(* LS Electric XG5000 project: PLC_Playground *)
(* PLC PlaygroundPLC *)

PROGRAM Main (* task: Scan Program *)
VAR
    I_Start AT %IX0.0.0 : BOOL;
    I_Stop AT %IX0.0.1 : BOOL;
    O_Run AT %QX0.0.0 : BOOL;
END_VAR
VAR
    _e1 : R_TRIG;
    _e2 : R_TRIG;
END_VAR

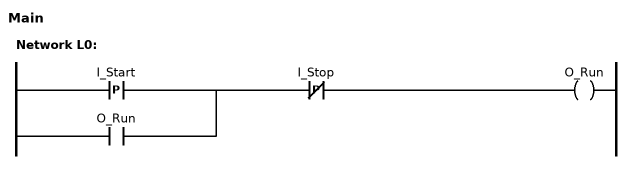
(* Rung L0 *)
_e1(CLK := I_Start);
_e2(CLK := I_Stop);
O_Run := (_e1.Q OR O_Run) AND NOT _e2.Q;
END_PROGRAM

PROGRAM FwdBwdMotor (* task: Scan Program *)
VAR
    I_Btn_Start AT %IX0.0.0 : BOOL;
    I_Btn_Stop AT %IX0.0.1 : BOOL;
    I_Sel_Direction AT %IX0.0.2 : BOOL;
    M_Is_Fwd AT %MX1 : BOOL := 1;
    M_Is_Moving AT %MX0 : BOOL := 0;
    O_Move_Bwd AT %QX0.0.1 : BOOL;
    O_Move_Fwd AT %QX0.0.0 : BOOL;
END_VAR
VAR
    _e1 : R_TRIG;
    _e2 : R_TRIG;
END_VAR

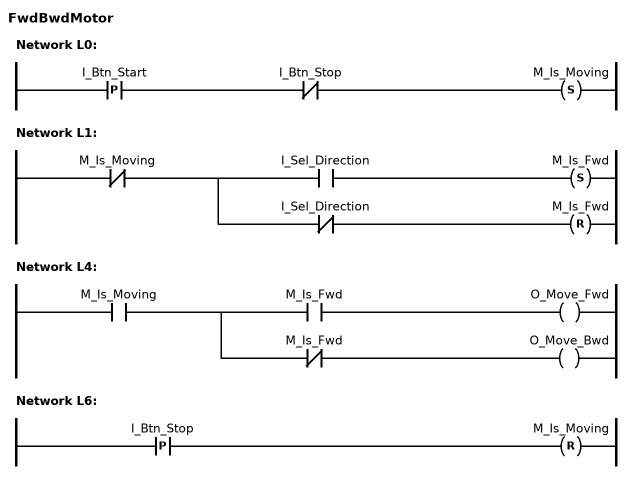
(* Rung L0 *)
_e1(CLK := I_Btn_Start);
IF _e1.Q AND NOT I_Btn_Stop THEN M_Is_Moving := TRUE; END_IF;
(* Rung L1 *)
IF NOT M_Is_Moving AND I_Sel_Direction THEN M_Is_Fwd := TRUE; END_IF;
IF NOT M_Is_Moving AND NOT I_Sel_Direction THEN M_Is_Fwd := FALSE; END_IF;
(* Rung L4 *)
O_Move_Fwd := M_Is_Moving AND M_Is_Fwd;
O_Move_Bwd := M_Is_Moving AND NOT M_Is_Fwd;
(* Rung L6 *)
_e2(CLK := I_Btn_Stop);
IF _e2.Q THEN M_Is_Moving := FALSE; END_IF;
END_PROGRAM

PROGRAM ButtonSequence (* task: Scan Program *)
VAR
    I_Btn_P1 AT %IX0.0.0 : BOOL;
    I_Btn_P2 AT %IX0.0.7 : BOOL;
    I_Btn_P3 AT %IX0.0.2 : BOOL;
    I_Btn_Ps AT %IX0.0.3 : BOOL;
    M_P1_WasPressed AT %MX0 : BOOL;
    M_P2_WasPressed AT %MX1 : BOOL;
    O_KM1 AT %QX0.0.0 : BOOL;
    O_Run AT %QX0.0.1 : BOOL;
END_VAR

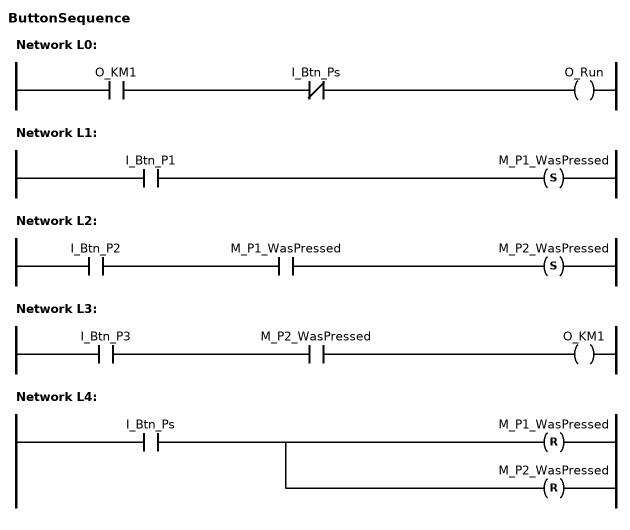
(* Rung L0 *)
O_Run := O_KM1 AND NOT I_Btn_Ps;
(* Rung L1 *)
IF I_Btn_P1 THEN M_P1_WasPressed := TRUE; END_IF;
(* Rung L2 *)
IF I_Btn_P2 AND M_P1_WasPressed THEN M_P2_WasPressed := TRUE; END_IF;
(* Rung L3 *)
O_KM1 := I_Btn_P3 AND M_P2_WasPressed;
(* Rung L4 *)
IF I_Btn_Ps THEN
    M_P1_WasPressed := FALSE;
    M_P2_WasPressed := FALSE;
END_IF;
END_PROGRAM